Fanuc KAREL source: get_CART_POS_fromRoki.kl

PROGRAM z_CART_POS
----------------------------------------------------
-- Creation date: 2021.11.01
-- Created by: ME
----------------------------------------------------
-- Version: v1
-- Modified from: HTTP1
----------------------------------------------------
-- Function:
----------------------------------------------------
-- Last modified: 2021.11.01
-- Last modified by: ME
------------
----------------------------------------
%NOLOCKGROUP
%ENVIRONMENT  REGOPE
--%TPMOTION
--%ENVIRONMENT MOTN
--%ENVIRONMENT MULTI
%ENVIRONMENT  STRNG
%COMMENT = 'getPOS_from_zRoki'
%NOABORT=ERROR+COMMAND
%NOPAUSE=ERROR+COMMAND+TPENABLE
%ALPHABETIZE
%INCLUDE KLEVKEYS
%INCLUDE KLEVKMSK
%INCLUDE KLEVCCDF
%INCLUDE KLIOUOP
%INCLUDE KLIOTYPS

CONST
    ROBOT_Config= 'NUT'
    SUCCESS = 0
    SNAP_REG = 199
    cc_SUCCESS =0
VAR
    id,XX,YY,ZZ,WW,PP,RR: STRING[10] --request params
    con: CONFIG
    x,y,z,w,p,r:  REAL
    temp_pos: XYZWPR
    HTTP_res_var : FILE
    HTTP_Res: STRING[20]
   STATUS,reg_ID, entry: INTEGER
    UFRAME,UTOOL: POSITION

----------------------------------------------------
-- BEGIN MyProgram
----------------------------------------------------

BEGIN
    -- clear the TPERROR screen
	--FORCE_SPMENU(TP_PANEL,SPI_TPUSER,1)
	WRITE(CHR(137),CHR(128))
	WRITE TPERROR(CHR(128))
   	WRITE('[X] Waiting for HTTP Req...',CR)

	    --set file for HTTP response
	    IF UNINIT(HTTP_Res) THEN
	        HTTP_Res='TD:RESPONSE.HTM'
	        WRITE('[X] INSIDE',CR)
	    ENDIF

	    WRITE('[X-GPOS] Openign File...',CR)
	    OPEN FILE HTTP_res_var ('RW', HTTP_Res)

	    --File open is a success or not
	    IF IO_STATUS(HTTP_res_var) = cc_SUCCESS THEN
	    	WRITE('[X-GPOS] OK',CR)
	       -- get Uframe and tframe for which reachiability of a position examine
	       GET_VAR(entry, '*SYSTEM*', '$MNUFRAME[1,1]', UFRAME, STATUS)
	       GET_VAR(entry, '*SYSTEM*', '$MNUTOOL[1,4]', UTOOL, STATUS)
	    	CNV_STR_INT(id,reg_ID)
		CNV_STR_REAL(XX,x)
		CNV_STR_REAL(YY,y)
		CNV_STR_REAL(ZZ,z)
		CNV_STR_REAL(WW,w)
		CNV_STR_REAL(PP,p)
		CNV_STR_REAL(RR,r)
	 	CNV_STR_CONF(ROBOT_Config,con,STATUS)
	 	temp_pos = POS(x,y,z,w,p,r,con)
	    	WRITE('[X] ',temp_pos,CR)
	        --I excluded Group number as i am having stackoverflow error
	         CHECK_EPOS(temp_pos,UFRAME,UTOOL,STATUS)
	         WRITE('[X] CHECK_EPOS',STATUS,CR)
	         --triger camera cycle if point not reachable
                IF STATUS <> cc_SUCCESS THEN
                	POST_ERR(STATUS, '1', 0, 0)
                	WRITE HTTP_res_var (400,CR)
                	SET_INT_REG(SNAP_REG,1,STATUS)
                    WRITE('PR values are not updated...',CR)
                    WRITE ('[X-GPOS] Operation is not SUCCESSFULL',CR)
                    WRITE ('[X-GPOS] Closing File...',CR)
                ELSE
                	SET_POS_REG(reg_ID,temp_pos,status,1)
                	WRITE HTTP_res_var (200,CR)
                     WRITE('PR values updated...',CR)
                     WRITE ('[X-GPOS] Operation is cc_SUCCESSFULL',CR)
                     WRITE ('[X-GPOS] Closing File...',CR)
                ENDIF
                CLOSE FILE HTTP_res_var
	    ELSE
		    WRITE ('[X-GPOS] File Operation isnot cc_SUCCESSFULL',CR)
		    CLOSE FILE HTTP_res_var
	    ENDIF

END z_CART_POS


    --IF status =0 THEN
        --WRITE('[X] Openign File...',CR)
        --OPEN FILE HTTP_res_var ('RW', HTTP_Res)
        --WRITE HTTP_res_var ('[X] OK',CR)
        ----I excluded Group number as i am having stackoverflow error
         --CHECK_EPOS(lpos,UFRAME,UTOOL,STATUS)
         --WRITE('[X] CHECK_EPOS',STATUS,CR)
         ----triger camera cycle if point not reachable
         --IF STATUS <> cc_SUCCESS THEN
         	--POST_ERR(STATUS, '1', 0, 0)
         	--WRITE HTTP_res_var (400,CR)
         	--SET_INT_REG(SNAP_REG,1,STATUS)
             --WRITE('PR values are not updated...',CR)
             --WRITE ('[X-GPOS] Operation is not SUCCESSFULL',CR)
             --WRITE ('[X-GPOS] Closing File...',CR)
         --ELSE
	          	--SET_POS_REG(reg_ID,temp_pos,status,1)
	         	--WRITE HTTP_res_var (200,CR)
	              --WRITE('PR values updated...',CR)
	              --WRITE ('[X-GPOS] Operation is cc_SUCCESSFULL',CR)
	              --WRITE ('[X-GPOS] Closing File...',CR)
         --ENDIF
        	--CLOSE FILE HTTP_res_var
        --
        ----undating position register
        --SET_POS_REG(reg_ID,temp_pos,status,1)
        --IF status <> SUCCESS THEN
            ----SET_INT_REG(REG_NUM, 1, status)
            --WRITE HTTP_res_var ('[X] PR values updated....',CR)
        --ENDIF
--
        --WRITE HTTP_res_var ('[X] Operation is SUCCESSFULL',CR)
        --WRITE HTTP_res_var ('[X] Closing File...',CR)
        --CLOSE FILE HTTP_res_var
    --ENDIF
